(* CoDeSys 2.3 export: _homeHeatingPlatform.rep *)
(* Libraries: STANDARD.LIB 5.6.98 11:03:02 *)

(* Task configuration *)
TASK Standard (PRIORITY := 0, INTERVAL := T#10ms);
END_TASK

(* Global variable list: ''/'Global_Variables' *)
VAR_GLOBAL CONSTANT
	ERROR_MARGIN : LREAL :=  1E-9;
END_VAR

(* Data type in '' *)
TYPE E_SimState :
(
	SimState_Initializing,
	SimState_Calculating,
	SimState_Stable
);
END_TYPE

(* POU '/_TestSuite/Simulation/HomeHeatingSim/BASEBLOCKS'/FB_BoilerSim, ST *)
FUNCTION_BLOCK FB_BoilerSim
VAR_INPUT
END_VAR
VAR_OUTPUT
END_VAR
VAR
END_VAR
;
END_FUNCTION_BLOCK

(* POU '/_TestSuite/Simulation/HomeHeatingSim/BASEBLOCKS'/FB_BurnerSim, ST *)
FUNCTION_BLOCK FB_BurnerSim
VAR_INPUT
	bOperatingOk: BOOL := TRUE;
END_VAR
VAR_OUTPUT
	bHasChanged : BOOL := FALSE;
	bIsOn: BOOL := FALSE;
END_VAR
VAR
	bInit: BOOL := TRUE;
	bOldState: BOOL := FALSE;
	Q_On  AT %I* : BOOL ;
	I_FlameDetected  AT %Q* : BOOL ;
END_VAR
IF bInit THEN
	bInit := FALSE;
	(* Do simulation initialization stuff *)
ELSE
	bHasChanged := FALSE;

	(*Do simulation running stuff *)
	IF bOperatingOk THEN
		bIsOn := Q_On;
	END_IF
	I_FlameDetected := bIsOn;

	bHasChanged := bOldState = NOT bIsOn;
	bOldState := bIsOn;
	(* If simulation calculations resulted in changes: bHasChanged := TRUE;  *)

	IF bIsOn THEN
		(*Do additional simulation*)
		;
	END_IF
END_IF
END_FUNCTION_BLOCK

(* POU '/_TestSuite/Simulation/HomeHeatingSim/BASEBLOCKS'/FB_FlowSensorSim, ST *)
FUNCTION_BLOCK FB_FlowSensorSim
VAR_INPUT
	bOperatingOk: BOOL := TRUE;
	lrFlow : LREAL;
	lrConversionFactor : LREAL := 0.01;
END_VAR
VAR_OUTPUT
	bHasChanged : BOOL := FALSE;
END_VAR
VAR
	bInit: BOOL := TRUE;
	I_value	AT %Q* : INT ;
END_VAR
IF bInit THEN
	bInit := FALSE;
	(* Do simulation initialization stuff *)
ELSE
	bHasChanged := FALSE;

	(*Do simulation running stuff *)
	I_value := REAL_TO_INT(  lrFlow / lrConversionFactor );

	(* If simulation calculations resulted in changes: bHasChanged := TRUE;  *)
	bHasChanged := TRUE;

END_IF
END_FUNCTION_BLOCK

(* POU '/_TestSuite/Simulation/HomeHeatingSim/BASEBLOCKS'/FB_HeatingUnitSim, ST *)
FUNCTION_BLOCK FB_HeatingUnitSim
VAR_INPUT
END_VAR
VAR_OUTPUT
END_VAR
VAR
END_VAR
;
END_FUNCTION_BLOCK

(* POU '/_TestSuite/Simulation/HomeHeatingSim/BASEBLOCKS'/FB_ManuallyValveSim, ST *)
FUNCTION_BLOCK FB_ManuallyValveSim
VAR_INPUT
	bOpen : BOOL := FALSE;
	bOperatingOk: BOOL := TRUE;
END_VAR
VAR_OUTPUT
	bHasChanged : BOOL := FALSE;
	bIsOpen: BOOL;
END_VAR
VAR
	bInit: BOOL := TRUE;
	bOldState: BOOL := FALSE;
END_VAR
IF bInit THEN
	bInit := FALSE;
	(* Do simulation initialization stuff *)
ELSE
	bHasChanged := FALSE;

	(*Do simulation running stuff *)
	bIsOpen := bOpen;

	bHasChanged := bOldState = NOT bIsOpen;
	bOldState := bIsOpen;
	(* If simulation calculations resulted in changes: bHasChanged := TRUE;  *)

	IF bIsOpen THEN
		(*Do additional simulation*)
		;
	END_IF
END_IF
END_FUNCTION_BLOCK
ACTION Close:
bOpen := FALSE;
END_ACTION
ACTION Open:
bOpen := TRUE;
END_ACTION

(* POU '/_TestSuite/Simulation/HomeHeatingSim/BASEBLOCKS'/FB_NormallyClosedValveSim, ST *)
FUNCTION_BLOCK FB_NormallyClosedValveSim
VAR_INPUT
	bOperatingOk: BOOL := TRUE;
END_VAR
VAR_OUTPUT
	bHasChanged : BOOL := FALSE;
	bIsOpen: BOOL;
END_VAR
VAR
	bInit: BOOL := TRUE;
	bOldState: BOOL := FALSE;
	Q_ControlValveSetpoint  AT %I* : BOOL ;
	I_ControValveFeedback AT %Q* : BOOL;
END_VAR
IF bInit THEN
	bInit := FALSE;
	(* Do simulation initialization stuff *)
ELSE
	bHasChanged := FALSE;

	(*Do simulation running stuff *)
	IF bOperatingOk THEN
		bIsOpen := Q_ControlValveSetpoint;
	END_IF

	bHasChanged := bOldState = NOT bIsOpen;
	bOldState := bIsOpen;
	(* If simulation calculations resulted in changes: bHasChanged := TRUE;  *)

	IF bIsOpen THEN
		(*Do additional simulation*)
		;
	END_IF

	I_ControValveFeedback := bIsOpen;
END_IF
END_FUNCTION_BLOCK

(* POU '/_TestSuite/Simulation/HomeHeatingSim/BASEBLOCKS'/FB_PipeSim, ST *)
FUNCTION_BLOCK FB_PipeSim
VAR_INPUT
	bOperatingOk: BOOL := TRUE;
END_VAR
VAR_OUTPUT
	bHasChanged : BOOL := FALSE;
END_VAR
VAR
	bInit : BOOL := TRUE;
END_VAR
IF bInit THEN
	bInit := FALSE;
	(* Do simulation initialization stuff *)
ELSE
	bHasChanged := FALSE;

	(*Do simulation running stuff *)
	(* If simulation calculations resulted in changes: bHasChanged := TRUE;  *)
END_IF
END_FUNCTION_BLOCK

(* POU '/_TestSuite/Simulation/HomeHeatingSim/BASEBLOCKS'/FB_PumpSim, ST *)
FUNCTION_BLOCK FB_PumpSim
VAR_INPUT
	bOperatingOk: BOOL := TRUE;
END_VAR
VAR_OUTPUT
	bHasChanged : BOOL := FALSE;
	bIsOn: BOOL := FALSE;
END_VAR
VAR
	bInit: BOOL := TRUE
;	bOldState: BOOL := FALSE;
	Q_On  AT %I* : BOOL ;
	I_OnFeedback  AT %Q* : BOOL ;
END_VAR
IF bInit THEN
	bInit := FALSE;
	(* Do simulation initialization stuff *)
ELSE
	bHasChanged := FALSE;

	(*Do simulation running stuff *)
	IF bOperatingOk THEN
		bIsOn := Q_On;
	END_IF

	bHasChanged := bOldState = NOT bIsOn;
	bOldState := bIsOn;
	(* If simulation calculations resulted in changes: bHasChanged := TRUE;  *)

	IF bIsOn THEN
		(*Do additional simulation*)
		;
	END_IF

	I_OnFeedback := bIsOn;
END_IF
END_FUNCTION_BLOCK

(* POU '/_TestSuite/Simulation/HomeHeatingSim/BASEBLOCKS'/FB_RadiatorSim, ST *)
FUNCTION_BLOCK FB_RadiatorSim
VAR_INPUT
END_VAR
VAR_OUTPUT
END_VAR
VAR
END_VAR
;
END_FUNCTION_BLOCK

(* POU '/_TestSuite/Simulation/HomeHeatingSim/BASEBLOCKS'/FB_SpeedSensorSim, ST *)
FUNCTION_BLOCK FB_SpeedSensorSim
VAR_INPUT
	bOperatingOk: BOOL := TRUE;
	lrRPM : LREAL := 0.0;
	lrConversionFactor : LREAL := 1.0;
END_VAR
VAR_OUTPUT
	bHasChanged : BOOL := FALSE;
END_VAR
VAR
	bInit: BOOL;
	I_value	AT %Q* : INT ;
END_VAR
IF bInit THEN
	bInit := FALSE;
	(* Do simulation initialization stuff *)
ELSE
	bHasChanged := FALSE;

	(*Do simulation running stuff *)
	I_value :=REAL_TO_INT(  lrRPM /  lrConversionFactor );

	(* If simulation calculations resulted in changes: bHasChanged := TRUE;  *)
	bHasChanged := TRUE;
END_IF
END_FUNCTION_BLOCK

(* POU '/_TestSuite/Simulation/HomeHeatingSim/BASEBLOCKS'/FB_TemperatureSensorSim, ST *)
FUNCTION_BLOCK FB_TemperatureSensorSim
VAR_INPUT
	bOperatingOk: BOOL := TRUE;
	lrTemperature : LREAL;
	lrConversionFactor : LREAL := 0.1;
END_VAR
VAR_OUTPUT
	bHasChanged : BOOL := FALSE;
END_VAR
VAR
	bInit: BOOL := TRUE;
	I_value	AT %Q* : INT ;
END_VAR
IF bInit THEN
	bInit := FALSE;
	(* Do simulation initialization stuff *)
ELSE
	bHasChanged := FALSE;

	(*Do simulation running stuff *)
	I_value := REAL_TO_INT( lrTemperature / lrConversionFactor );

	(* If simulation calculations resulted in changes: bHasChanged := TRUE;  *)
	bHasChanged := TRUE;
END_IF
END_FUNCTION_BLOCK

(* POU '/_TestSuite/Simulation/HomeHeatingSim/BASEBLOCKS'/FB_ThermostatSim, ST *)
FUNCTION_BLOCK FB_ThermostatSim
VAR_INPUT
	bOperatingOk: BOOL := TRUE;
	lrRoomTemperature : LREAL;
	lrRequestedTemperature: LREAL;
	lrConversionFactor : LREAL := 0.1;
END_VAR
VAR_OUTPUT
	bHasChanged : BOOL := FALSE;
END_VAR
VAR
	bInit: BOOL := TRUE;
	I_requestedTemp	AT %Q* : INT ;
	I_roomTemp	AT %Q* : INT ;
END_VAR
IF bInit THEN
	bInit := FALSE;
	(* Do simulation initialization stuff *)
ELSE
	bHasChanged := FALSE;

	(*Do simulation running stuff *)
	I_requestedTemp := REAL_TO_INT( lrRequestedTemperature / lrConversionFactor );
	I_roomTemp := REAL_TO_INT(  lrRoomTemperature / lrConversionFactor );

	(* If simulation calculations resulted in changes: bHasChanged := TRUE;  *)
	bHasChanged := TRUE;
END_IF
END_FUNCTION_BLOCK

(* POU '/_TestSuite/Simulation/HomeHeatingSim/BASEBLOCKS'/FB_ThreeValveSim, ST *)
FUNCTION_BLOCK FB_ThreeValveSim
VAR_INPUT
	bOperatingOk: BOOL := TRUE;
END_VAR
VAR_OUTPUT
	bHasChanged : BOOL := FALSE;
	iPosition : INT :=0; (*0=Mid, 1=Left, 2=Right*)
	bThreeValveLeft  : BOOL ;
	bThreeValveRight : BOOL ;
	bThreeValveOpen: BOOL;
END_VAR
VAR
	bInit: BOOL := TRUE;
	iOldPosition : INT :=0; (*0=Mid, 1=Left, 2=Right*)

	Q_ThreeValveSetpoint  AT %I* : INT;
	I_ThreeValveFeedback AT %Q* : INT;
END_VAR
IF bInit THEN
	bInit := FALSE;
	(* Do simulation initialization stuff *)
ELSE
	bHasChanged := FALSE;

	(*Do simulation running stuff *)
	(* Allow for injecting fault conditions*)
	IF bOperatingOk THEN
		iPosition := Q_ThreeValveSetpoint;
	END_IF

	bHasChanged := iOldPosition <> iPosition;
	iOldPosition := iPosition;
	(* If simulation calculations resulted in changes: bHasChanged := TRUE;  *)

	I_ThreeValveFeedback := iPosition;
	bThreeValveLeft := (iPosition <> 2);
	bThreeValveRight := (iPosition <> 1);
	bThreeValveOpen :=  TRUE;
END_IF
END_FUNCTION_BLOCK

(* POU '/HOMEHEATING/BASEBLOCKS'/FB_Boiler, ST *)
FUNCTION_BLOCK FB_Boiler
VAR_INPUT
	bWarmUp : BOOL := FALSE;
END_VAR
VAR_OUTPUT
	lrTempSetpointLow : LREAL := 85.0;
	lrTempSetpointHigh : LREAL := 90.0;

END_VAR
VAR
END_VAR
;
END_FUNCTION_BLOCK
ACTION DontWarmUp:
bWarmUp := FALSE;
END_ACTION
ACTION DoWarmUp:
bWarmUp := TRUE;
END_ACTION

(* POU '/HOMEHEATING/BASEBLOCKS'/FB_Burner, ST *)
FUNCTION_BLOCK FB_Burner
VAR_INPUT
(* Change to setpoint in percentage *)
	bOn : BOOL := FALSE;
	bHeatRequested : BOOL := FALSE;
END_VAR
VAR_OUTPUT
	bFlameDetected : BOOL := FALSE;
END_VAR
VAR
	Q_On  AT %Q* : BOOL ;
	I_FlameDetected  AT %I* : BOOL ;
END_VAR
Q_On := bOn;
bFlameDetected := I_FlameDetected;
END_FUNCTION_BLOCK
ACTION Off:
bOn := FALSE;
END_ACTION
ACTION On:
bOn := TRUE;
END_ACTION

(* POU '/HOMEHEATING/BASEBLOCKS'/FB_FlowSensor, ST *)
FUNCTION_BLOCK FB_FlowSensor
VAR_INPUT
	lrConversionFactor : LREAL := 0.01;
END_VAR
VAR_OUTPUT
	lrFlow : LREAL;
END_VAR
VAR
	I_value	AT %I* : INT ;
END_VAR
lrFlow := I_value * lrConversionFactor;
END_FUNCTION_BLOCK

(* POU '/HOMEHEATING/BASEBLOCKS'/FB_ManuallyValve, ST *)
FUNCTION_BLOCK FB_ManuallyValve
VAR_INPUT
END_VAR
VAR_OUTPUT
END_VAR
VAR
END_VAR
;
END_FUNCTION_BLOCK

(* POU '/HOMEHEATING/BASEBLOCKS'/FB_NormallyClosedValve, ST *)
FUNCTION_BLOCK FB_NormallyClosedValve
VAR_INPUT
	bOpen : BOOL := FALSE;
END_VAR
VAR_OUTPUT
	bOpenFeedback : BOOL;
END_VAR
VAR
	Q_ControlValveSetpoint  AT %Q* : BOOL ; (* True = Open*)
	I_ControValveFeedback AT %I* : BOOL;
END_VAR
Q_ControlValveSetpoint := bOpen;

(* Provide some feedback *)
bOpenFeedback := I_ControValveFeedback;
END_FUNCTION_BLOCK
ACTION Close:
bOpen := FALSE;
END_ACTION
ACTION Open:
bOpen := TRUE;
END_ACTION

(* POU '/HOMEHEATING/BASEBLOCKS'/FB_Pump, ST *)
FUNCTION_BLOCK FB_Pump
VAR_INPUT
	bOn : BOOL := FALSE;
END_VAR
VAR_OUTPUT
	bOnFeedback : BOOL := FALSE;
END_VAR
VAR
	Q_On  AT %Q* : BOOL ;
	I_OnFeedback  AT %I* : BOOL ;
END_VAR
Q_On := bOn;

(* Provide some feedback *)
bOnFeedback := I_OnFeedback;
END_FUNCTION_BLOCK
ACTION Off:
bOn := FALSE;
END_ACTION
ACTION On:
bOn := TRUE;
END_ACTION

(* POU '/HOMEHEATING/BASEBLOCKS'/FB_Radiator, ST *)
FUNCTION_BLOCK FB_Radiator
VAR_INPUT
	bWarmUp : BOOL := FALSE;
END_VAR
VAR_OUTPUT
END_VAR
VAR
END_VAR
;
END_FUNCTION_BLOCK
ACTION DontWarmUp:
bWarmUp := FALSE;
END_ACTION
ACTION DoWarmUp:
bWarmUp := TRUE;
END_ACTION

(* POU '/HOMEHEATING/BASEBLOCKS'/FB_SpeedSensor, ST *)
FUNCTION_BLOCK FB_SpeedSensor
VAR_INPUT
	lrConversionFactor : LREAL := 1.0;
END_VAR
VAR_OUTPUT
	lrRPM : LREAL := 0.0;
END_VAR
VAR
	I_value	AT %I* : INT ;
END_VAR
lrRPM := I_value * lrConversionFactor;
END_FUNCTION_BLOCK

(* POU '/HOMEHEATING/BASEBLOCKS'/FB_TemperatureSensor, ST *)
FUNCTION_BLOCK FB_TemperatureSensor
VAR_INPUT
	lrConversionFactor : LREAL := 0.1;
END_VAR
VAR_OUTPUT
	lrTemperature : LREAL;
END_VAR
VAR
	I_value	AT %I* : INT ;
END_VAR
lrTemperature := I_value * lrConversionFactor;
END_FUNCTION_BLOCK

(* POU '/HOMEHEATING/BASEBLOCKS'/FB_Thermostat, ST *)
FUNCTION_BLOCK FB_Thermostat
VAR_INPUT
	lrConversionFactor: LREAL := 0.1;
END_VAR
VAR_OUTPUT
	lrRequestedTemperature: LREAL;
	lrRoomTemperature: LREAL;
	lrTempSetpointLow : LREAL;
	lrTempSetPointHigh : LREAL;
END_VAR
VAR
	lrHysteresis : LREAL := 0.5;
	I_requestedTemp	AT %I* : INT ;
	I_roomTemp	AT %I* : INT ;
END_VAR
lrRoomTemperature :=I_roomTemp * lrConversionFactor;
lrRequestedTemperature :=I_requestedTemp * lrConversionFactor;
lrTempSetpointLow := lrRequestedTemperature - lrHysteresis;
lrTempSetpointHigh := lrRequestedTemperature + lrHysteresis;
END_FUNCTION_BLOCK

(* POU '/HOMEHEATING/BASEBLOCKS'/FB_ThreeValve, ST *)
FUNCTION_BLOCK FB_ThreeValve
VAR_INPUT
	iPositionSetpoint : INT :=0; (*0=Mid, 1=Left, 2=Right*)
END_VAR
VAR_OUTPUT
	bThreeValveLeft  : BOOL ;
	bThreeValveRight : BOOL ;
	bThreeValveBoth: BOOL;
END_VAR
VAR
	iPositionFeedback : INT := 0;
	Q_ThreeValveSetpoint  AT %Q* : INT;
	I_ThreeValveFeedback AT %I* : INT;
END_VAR
Q_ThreeValveSetpoint := iPositionSetpoint;
iPositionFeedback := I_ThreeValveFeedback;

(* Provide some feedback *)
bThreeValveLeft := (iPositionFeedback = 1);
bThreeValveRight := (iPositionFeedback = 2);
bThreeValveBoth :=  (iPositionFeedback = 0);
END_FUNCTION_BLOCK
ACTION OpenBoth:
iPositionSetpoint := 0;
END_ACTION
ACTION OpenLeft:
iPositionSetpoint := 1;
END_ACTION
ACTION OpenRight:
iPositionSetpoint := 2;
END_ACTION

(* POU '/INFRASTRUCTURE'/F_Assert, ST *)
(*****************************************************************
 Copyright Sioux Embedded Systems B.V. 
 All rights reserved.
******************************************************************)
FUNCTION F_Assert : BOOL
VAR_INPUT
	bCondition : BOOL := FALSE;
	text : STRING;
END_VAR
VAR
	a : INT := 1;
	b : INT := 0;
	c : INT := 0;
END_VAR
IF NOT bCondition THEN
	(*Deliberate Assert, See the Callstack: Online -> Call Stack*)
	c := a/b;
END_IF
F_Assert := FALSE;
END_FUNCTION

(* Visualisation HeatingSystem
70 more shapes without text or variables
*)
